PROGRAM MAIN
VAR
	// Variables established here, including Motor, Timer, and Output storage
	bMotorRun: BOOL := TRUE;
	
	tMinuteTimer: TON;
	
	nTotalMinutes: INT := 0;
	nTotalHours: INT := 0;
	
END_VAR

// TImer detects if motor is currently running and timer isn't already completed
tMinuteTimer(IN:= bMotorRun AND NOT tMinuteTimer.Q, PT:= T#5S);
// INT for Minutes counts up everytime the timer is completed and resets at 60 for the hourly conversion
// Ideally this could be applied to keep track of time in-between maintenance cycles.
IF tMinuteTimer.Q THEN
	nTotalMinutes := nTotalMinutes +1;
	IF nTotalMinutes = 60 THEN
		nTotalMinutes := 0;
		nTotalHours := nTotalHours + 1;
	END_IF;
END_IF;

END_PROGRAM

(* stored: Version 1.1.0.1, ProductVersion 3.1.4024.16
   POU MAIN: Id {be840c94-27f3-451b-a264-5caf577e0e52}, SpecialFunc None *)
